{attribute addProperty BoxType "EL3443-0000-0016"}
{attribute addProperty Id "VoltageAT %I*REAL32417CurrentAT %I*REAL32418"}
{attribute addProperty CRC "6145035"}
{attribute addProperty SizeInBites "64"}
{attribute addProperty SizeInBytes "8"}
TYPE L3_Basic_005DC40B :
STRUCT
	{attribute addProperty Name "Voltage"}
	Voltage AT %I* : REAL;
	{attribute addProperty Name "Current"}
	Current AT %I* : REAL;
END_STRUCT
END_TYPE

(* stored: Version 1.2.0.0, ProductVersion 3.1.4024.9
   DUT L3_Basic_005DC40B: Id {00497f61-ed02-466b-9918-56c2e62f6e5b} *)
